# EPICS autosave request: softGlueApp/Db/softGlue_config_settings.req
$(P)$(H)streamMux
$(P)$(H)FO9Mux
$(P)$(H)FO10Mux
$(P)$(H)FO11Mux
$(P)$(H)FO12Mux
